{attribute addProperty BoxType "EJ1914-0000-0017"}
{attribute addProperty Id "FSOEAT %Q*FSOE_27E40C71486"}
{attribute addProperty CRC "3800498592"}
{attribute addProperty SizeInBites "48"}
{attribute addProperty SizeInBytes "6"}
TYPE FSoE_Outputs_E28701A0 :
STRUCT
	{attribute addProperty Name "FSOE"}
	FSOE AT %Q* : FSOE_27E40C71;
END_STRUCT
END_TYPE

(* stored: Version 1.2.0.0, ProductVersion 3.1.4024.9
   DUT FSoE_Outputs_E28701A0: Id {9842e881-133c-453e-924d-88918e5f762d} *)
